(* Ansteuerprogramm der Leitachse. Das Programm hat die Aufgabe, 
   die Leitachse in eine Bewegung konstanter Ge-schwindigkeit zu versetzen, 
   wieder anzuhalten und im Falle eines Fehlers die Achse durch einen Reset 
   wieder in einen funktionstüchtigen Zustand zu versetzen. *)

PROGRAM MasterAnAus
VAR
	//stateMaster				: MoveState_t;		// Programmablauf über Zustandsvariable

	PowerMaster				: MC_Power;			// Schaltet Software-Freigabe der Leitachse
	PowerMasterOut			: ST_McOutputs;		// 
	
	ResetMaster				: MC_Reset;			// Setzt Achsfehler zurück
	ResetMasterOut			: ST_McOutputs;	
	
	MoveMaster 				: MC_MoveVelocity;	// Versetzt Leitachse in Bewegung konstanter Geschwindigkeit
	MoveMasterOut			: ST_McOutputs;
	
	HaltMaster				: MC_Halt;			// Hält Leitachse an
	HaltMasterOut			: ST_McOutputs;
	startMasterTrig: R_TRIG;
	MoveNewMaster: MC_MoveVelocity;
	MoveNewMasterOut: ST_McOutputs;
	stateMaster: Movestate_t;
END_VAR

//startMasterTrig(clk := AbwicklerStart);
GlobaleVariablen.Master();

CASE stateMaster OF
(* ===========================================================================================
   Zustand 1: Programm ist im Ausgangszustand und wartet auf Benutzereingabe. Alle 
   Funktionsbausteine werden initialisiert, etwaige Fehler zurückgesetzt. *)
	MOVESTATE_INIT :
		MoveMaster.Execute := FALSE;
		MoveNewMaster.Execute := FALSE;
		ResetMaster.Execute := FALSE;
		HaltMaster.Execute := FALSE;
		PowerMaster.Enable := FALSE;
		PowerMaster.Enable_Positive := FALSE;
		MasterLaeuft := FALSE;
		IF MasterStart THEN
			stateMaster := MOVESTATE_ENABLE;
		END_IF

(* ===========================================================================================
   Zustand 2: Schlalten der allgemeinen Software-Freigabe, Vorschubfreigabe in positive Richtung
   durch MC_Power. Sobald Funktionsbaustein MC_Power die Betriebsbereitschaft der Achse signalisiert,
   Zustandsübergang in Forward*)
	MOVESTATE_ENABLE :
		PowerMaster.Enable := TRUE;
		IF PowerMaster.Status THEN
			stateMaster := MOVESTATE_FORWARD;
		ELSIF PowerMaster.Error THEN
			stateMaster := MOVESTATE_ERROR;
		END_IF
		
(* ===========================================================================================
   Zustand 3: Starten des Mastern in positive Richtung mit konstanter Geschwindigkeit. 
   Zustandsübergang durch Bedienerbefehl.*)		
	MOVESTATE_FORWARD :
	
		MoveMaster.Execute := TRUE;

		IF alt_xPunkt >= 0 THEN
			MoveMaster.Direction := MC_Positive_Direction;
			MoveMaster.Velocity := GlobaleVariablen.alt_xPunkt;
		ELSIF alt_xPunkt < 0 THEN
			MoveMaster.Direction := MC_Negative_Direction;
			MoveMaster.Velocity := (-1) * GlobaleVariablen.alt_xPunkt;
		ELSE MoveMaster.Direction := MC_Undefined_Direction;
		END_IF
		IF MoveMasterOut.Active THEN
			MoveMaster.Execute := FALSE;
			MasterLaeuft := TRUE;
			stateMaster := MOVESTATE_NEW_FORWARD;
		END_IF
		IF MoveMasterOut.Done THEN
			MasterLaeuft := TRUE;
			MoveMaster.Execute := FALSE;
			stateMaster := MOVESTATE_FORWARD;
		END_IF
		IF MasterStopp THEN
			MoveMaster.Velocity := 0;
			AbwicklerStopp := TRUE;
			AbwicklerStart := FALSE;
			AufwicklerStopp := TRUE;
			AufwicklerStart := FALSE;
			IF AbwicklerLaeuft = FALSE AND AufwicklerLaeuft = FALSE THEN
				MasterStart := FALSE;
				stateMaster := MOVESTATE_STOPMASTER;
			END_IF
		END_IF
		IF MoveMaster.Error THEN
			stateMaster := MOVESTATE_ERROR;
		END_IF
		
	MOVESTATE_NEW_FORWARD:
		MoveNewMaster.Execute := TRUE;

		IF alt_xPunkt >= 0 THEN
			MoveNewMaster.Direction := MC_Positive_Direction;
			MoveNewMaster.Velocity := GlobaleVariablen.alt_xPunkt;
		ELSIF alt_xPunkt < 0 THEN
			MoveNewMaster.Direction := MC_Negative_Direction;
			MoveNewMaster.Velocity := (-1) * GlobaleVariablen.alt_xPunkt;
		ELSE MoveNewMaster.Direction := MC_Undefined_Direction;
		END_IF
		IF MoveNewMasterOut.Active THEN
			MoveNewMaster.Execute := FALSE;
			MasterLaeuft := TRUE;
			stateMaster := MOVESTATE_FORWARD;
		END_IF
		IF MoveNewMasterOut.Done THEN
			MoveNewMaster.Execute := FALSE;
			MasterLaeuft := TRUE;
			stateMaster := MOVESTATE_NEW_FORWARD;
		END_IF
		IF MasterStopp THEN
			MoveNewMaster.Velocity := 0;
			AbwicklerStopp := TRUE;
			AbwicklerStart := FALSE;
			AufwicklerStopp := TRUE;
			AufwicklerStart := FALSE;
			IF AbwicklerLaeuft = FALSE AND AufwicklerLaeuft = FALSE THEN
				MasterStart := FALSE;
				stateMaster := MOVESTATE_STOPMASTER;
			END_IF
		END_IF
		IF MoveNewMasterOut.Error THEN
			stateMaster := MOVESTATE_ERROR;
		END_IF
		
(* ===========================================================================================
   Zustand 4: Anhalten der Leitachse, im Anschluss Rückkehr in den Ausgangszustand. *)		
	MOVESTATE_STOPMASTER :
		
		IF HaltMaster.Done THEN
			MasterStopp := FALSE;
			HaltMaster.Execute := FALSE;
			MasterStart := FALSE;
			MasterLaeuft := FALSE;
			stateMaster := MOVESTATE_INIT;
		ELSE
			HaltMaster.Execute := TRUE;
		END_IF
		IF HaltMaster.Error OR HaltMaster.CommandAborted THEN
			HaltMaster.Execute := FALSE;
			stateMaster := MOVESTATE_ERROR;
		END_IF

(* ===========================================================================================
   Zustand 5: Im Falle eines Bausteinfehlers wird überprüft, ob sich die Achse ebenfalls im    
   Fehlerzustand befindet, was einen Achsreset erfordert. Andernfalls werden Bausteinfehler 
   im Zustand Init zurückgesetzt.*)		
	MOVESTATE_ERROR :
		IF Master.Status.Error THEN
			stateMaster := MOVESTATE_RESET;	// Reset bei Achsfehler
		ELSE
			stateMaster := MOVESTATE_INIT;	// Funktionsbausteinfehler erfordert keinen Reset
		END_IF

(* ===========================================================================================
   Zustand 6:  Durchführung des Achsreset im Fehlerfall  *)		
	MOVESTATE_RESET :
		MasterStopp := FALSE;
		ResetMaster.Execute := TRUE;
		IF ResetMaster.Done THEN
			stateMaster := MOVESTATE_INIT;
		ELSIF ResetMaster.Error THEN
			stateMaster := MOVESTATE_INIT; (* Falls Reset nicht gelingt, Benutzereingriff erforderlich *)
		END_IF
		
END_CASE

// Zyklusmäßige Aufrufe
ActPower();		// Aufruf des Power Funktionsbausteines
ActMove();		// Aufruf des Move-Funktionsbausteines
ActReset();		// Aufruf des Reset-Funktionsbausteines

ACTION ActMove:
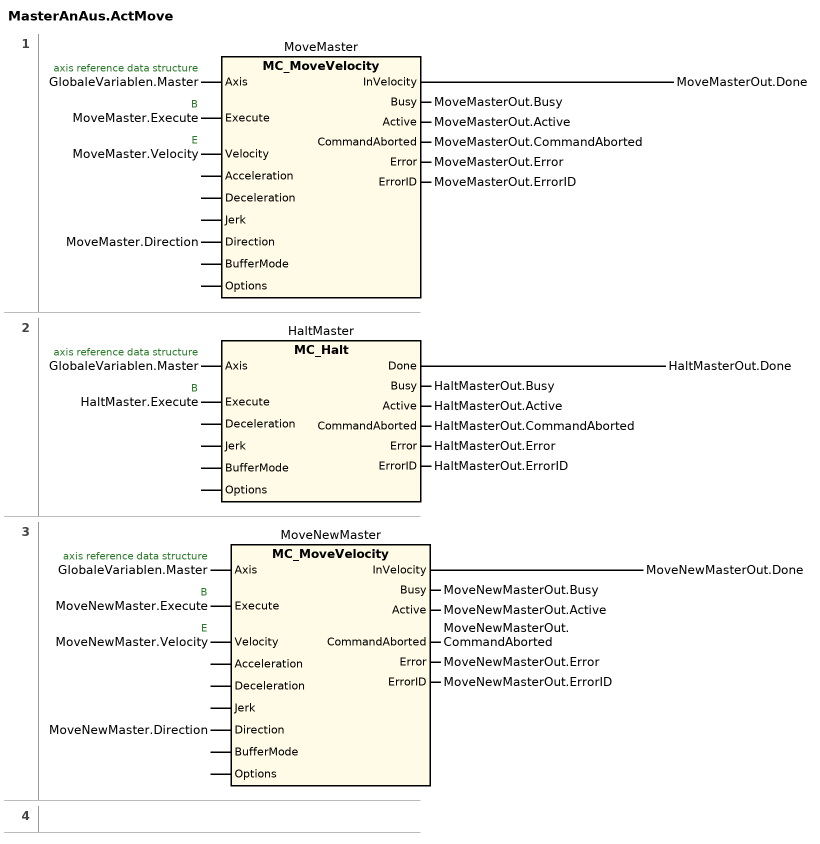
// NETWORK 1
//   GlobaleVariablen.Master: axis reference data structure
//   MoveMaster.Execute: B
//   MoveMaster.Velocity: E
MoveMaster(
    Axis := GlobaleVariablen.Master,
    Execute := MoveMaster.Execute,
    Velocity := MoveMaster.Velocity,
    Direction := MoveMaster.Direction,
    Busy => MoveMasterOut.Busy,
    Active => MoveMasterOut.Active,
    CommandAborted => MoveMasterOut.CommandAborted,
    Error => MoveMasterOut.Error,
    ErrorID => MoveMasterOut.ErrorID); // MC_MoveVelocity
MoveMasterOut.Done := MoveMaster.InVelocity;

// NETWORK 2
//   GlobaleVariablen.Master: axis reference data structure
//   HaltMaster.Execute: B
HaltMaster(
    Axis := GlobaleVariablen.Master,
    Execute := HaltMaster.Execute,
    Busy => HaltMasterOut.Busy,
    Active => HaltMasterOut.Active,
    CommandAborted => HaltMasterOut.CommandAborted,
    Error => HaltMasterOut.Error,
    ErrorID => HaltMasterOut.ErrorID); // MC_Halt
HaltMasterOut.Done := HaltMaster.Done;

// NETWORK 3
//   GlobaleVariablen.Master: axis reference data structure
//   MoveNewMaster.Execute: B
//   MoveNewMaster.Velocity: E
MoveNewMaster(
    Axis := GlobaleVariablen.Master,
    Execute := MoveNewMaster.Execute,
    Velocity := MoveNewMaster.Velocity,
    Direction := MoveNewMaster.Direction,
    Busy => MoveNewMasterOut.Busy,
    Active => MoveNewMasterOut.Active,
    CommandAborted => MoveNewMasterOut.CommandAborted,
    Error => MoveNewMasterOut.Error,
    ErrorID => MoveNewMasterOut.ErrorID); // MC_MoveVelocity
MoveNewMasterOut.Done := MoveNewMaster.InVelocity;

// NETWORK 4
END_ACTION

ACTION ActPower:
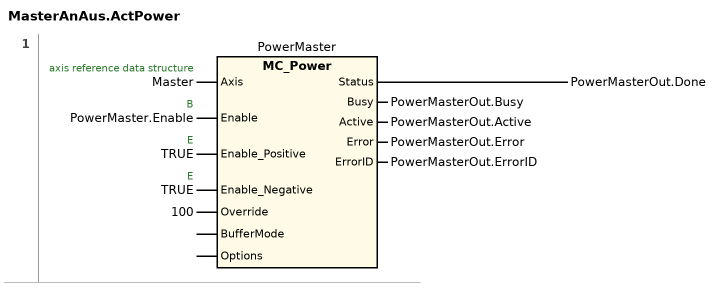
// NETWORK 1
//   Master: axis reference data structure
//   PowerMaster.Enable: B
//   TRUE: E
PowerMaster(
    Axis := Master,
    Enable := PowerMaster.Enable,
    Enable_Positive := TRUE,
    Enable_Negative := TRUE,
    Override := 100,
    Busy => PowerMasterOut.Busy,
    Active => PowerMasterOut.Active,
    Error => PowerMasterOut.Error,
    ErrorID => PowerMasterOut.ErrorID); // MC_Power
PowerMasterOut.Done := PowerMaster.Status;
END_ACTION

ACTION ActReset:
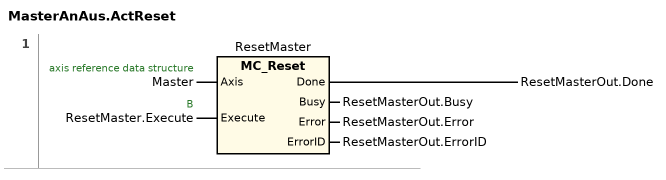
// NETWORK 1
//   Master: axis reference data structure
//   ResetMaster.Execute: B
ResetMaster(
    Axis := Master,
    Execute := ResetMaster.Execute,
    Busy => ResetMasterOut.Busy,
    Error => ResetMasterOut.Error,
    ErrorID => ResetMasterOut.ErrorID); // MC_Reset
ResetMasterOut.Done := ResetMaster.Done;
END_ACTION

END_PROGRAM

(* stored: Version 1.1.0.1, ProductVersion 3.1.4024.11
   POU MasterAnAus: Id {e8703064-222c-40b1-904c-3074ce7c59b7}, SpecialFunc None
   Action ActMove: Id {c7f6f98c-2816-41c3-b934-1024e7cb7466}
   Action ActPower: Id {a5b49902-28f4-4249-85a2-b70e23dde08b}
   Action ActReset: Id {02d780b9-f744-4898-a2e9-c26494de6f03} *)
